// TIA Portal V20 export
TYPE "typeSequenceControlNodeJobInterfaceCommands"
// stored: Namespace Unit1.Em6
   STRUCT
      spare { ExternalWritable := 'False'} : Bool;
   END_STRUCT;
END_TYPE
